FUNCTION_BLOCK Serialize

VAR_INPUT
	a : BYTE;
	b : LREAL;
	c : ARRAY[1..6, 1..6] OF LREAL;
END_VAR

VAR_OUTPUT
	sendbuffer : ARRAY[0..1023] OF BYTE;
END_VAR

VAR
	i, j : DINT;
	offset : UDINT := 0;
END_VAR

offset := 0;
MEMCPY(ADR(sendbuffer[offset]), ADR(a), SIZEOF(a));

offset := offset + SIZEOF(a);
MEMCPY(ADR(sendbuffer[offset]), ADR(b), SIZEOF(b));

offset := offset + SIZEOF(b);
FOR i := 1 TO 6 DO
	FOR j := 1 TO 6 DO
		MEMCPY(ADR(sendbuffer[offset]), ADR(c[i,j]), SIZEOF(c[i,j]));
		offset := offset + SIZEOF(b);
	END_FOR
END_FOR

END_FUNCTION_BLOCK

(* stored: Version 1.1.0.1, ProductVersion 3.1.4024.13
   POU Serialize: Id {80769f59-008c-4d60-ba2b-7737fa5de118}, SpecialFunc None *)
